# EPICS autosave request: measCompApp/Db/measCompTemperatureIn_settings.req
$(P)$(R)Scale
$(P)$(R)TCType
$(P)$(R)Filter
$(P)$(R).LOPR
$(P)$(R).HOPR
$(P)$(R).PREC
$(P)$(R).SCAN
